FUNCTION_BLOCK BaseConnector
VAR_INPUT
END_VAR
VAR_OUTPUT
END_VAR
VAR
END_VAR
VAR_STAT
	sp	: SymbolProvider;
END_VAR

END_FUNCTION_BLOCK

(* stored: Version 1.1.0.1, ProductVersion 3.1.4024.11
   POU BaseConnector: Id {a4e3b6d8-322f-496d-8bff-a7ec971249cd}, SpecialFunc None *)
